Yaskawa INFORM job: SKRZYNIA_4040_0_STOPNI_2OBR.JBI

/JOB
//NAME SKRZYNIA_4040_0_STOPNI_2OBR
///FOLDERNAME 02-SKRZYNIE_JOBS
//POS
///NPOS 466,466,0,38,0,0
///TOOL 0
///POSTYPE PULSE
///PULSE
C00000=1055,-24125,84372,288,19725,204
C00001=0,-15438,65714,0,-68532,0
C00002=4718,-16587,59952,3396,-65485,-935
C00003=32997,-21499,42555,27623,-61436,21376
C00004=31759,-20688,42932,26837,-60850,21559
C00005=28987,-21156,42712,24818,-60442,22222
C00006=33447,-21964,42352,27886,-61721,21330
C00007=37687,-23357,41794,30651,-63289,20620
C00008=38979,-19018,48057,32961,-64962,20678
C00009=37261,-18075,48526,31902,-64209,20901
C00010=35830,-17198,48994,31015,-63571,21092
C00011=34080,-17614,48768,29780,-63290,21485
C00012=37261,-18075,48526,31902,-64209,20901
C00013=47373,-21912,40596,41149,-66086,26950
C00014=45033,-20851,41104,39798,-65001,27223
C00015=42790,-19693,41704,38494,-63946,27495
C00016=41070,-20182,41442,37324,-63566,27891
C00017=45033,-20851,41104,39798,-65001,27223
C00018=59624,-29540,14278,64846,-60867,16042
C00019=59624,-29540,14278,64846,-60867,16042
C00020=57357,-28542,14780,63940,-59509,16120
C00021=56188,-29140,14476,63237,-58995,16387
C00022=59588,-29370,14363,64862,-60819,16012
C00023=70875,-38414,-12574,117781,-105744,5605
C00024=70875,-38414,-12574,117781,-105744,5605
C00025=58486,-39981,-10562,86359,-50427,5279
C00026=56769,-35832,-2792,84059,-49443,6631
C00027=55152,-35009,-2405,83835,-48426,6454
C00028=53661,-35722,-2740,83085,-47530,6682
C00029=56769,-35832,-2792,84059,-49443,6631
C00030=45044,-23015,37260,35797,-71879,25522
C00031=39973,-29571,18873,35060,-63052,24165
C00032=38620,-28701,19269,34339,-62304,24363
C00033=36409,-29254,19014,32896,-61805,24958
C00034=44451,-29039,21934,37281,-65892,23702
C00035=49472,-39353,6917,53118,-50908,20251
C00036=45058,-39356,3832,51653,-47640,20099
C00037=42883,-38319,4163,50577,-46309,20295
C00038=40255,-38926,3967,48502,-45334,21060
C00039=46774,-39679,3737,52663,-48537,19827
C00040=48708,-40455,3517,53615,-49689,19657
C00041=43798,-39237,3871,50850,-47027,20335
C00042=41951,-38324,4161,49930,-45891,20507
C00043=39836,-38844,3994,48234,-45126,21137
C00044=48489,-40338,3551,53521,-49551,19665
C00045=41144,-42823,8332,45214,-41270,16613
C00046=27655,-47386,17113,29958,-26061,11007
C00047=27657,-47383,17112,100898,-60101,11012
C00048=27657,-47383,17112,100898,-60101,11012
C00049=48489,-40338,3551,53521,-49551,19665
C00050=44432,-39026,3936,51363,-47247,20139
C00051=42487,-38069,4248,50403,-46050,20315
C00052=39061,-38795,4009,47695,-44769,21310
C00053=44432,-39026,3936,51363,-47247,20139
C00054=43521,-36748,12770,50182,-45701,23408
C00055=41846,-35383,13175,49516,-44517,23399
C00056=39971,-34448,13485,48491,-43408,23582
C00057=37453,-34980,13306,46330,-42542,24334
C00058=41846,-35383,13175,49516,-44517,23399
C00059=78369,-41260,16071,67181,-65880,21417
C00060=137,-45861,52341,97,-67596,-14
C00061=11549,-53044,26255,3918,7271,6746
C00062=11549,-23006,80296,3918,7271,6746
C00063=11549,-23006,80296,3918,7271,6746
C00064=57941,-59676,-5815,65032,-36778,-7179
C00065=75493,-63502,-64712,103874,-64610,-6298
C00066=48206,-58699,-62794,109567,-46310,-10557
C00067=43841,-59955,-65018,113836,-43076,-9157
C00068=55379,-67378,-68041,108237,-48773,-4935
C00069=60826,-65014,-65501,105394,-54241,-6755
C00070=28458,-37240,33167,37371,-31902,2053
C00071=0,-44704,54767,0,2714,0
C00072=1055,-24125,84372,288,19725,204
C00073=0,-15438,65714,0,-68532,0
C00074=0,-15438,65714,966,-70097,42926
C00075=69988,-9219,57065,61610,-82752,27767
C00076=63113,-6157,59685,58080,-79692,28271
C00077=46291,-7558,63674,40492,-74068,29264
C00078=49370,-5991,66013,43448,-75651,29403
C00079=53417,-8187,64183,45775,-77170,28968
C00080=63113,-6157,59685,58080,-79692,28271
C00081=69988,-9219,57065,61610,-82752,27767
C00082=0,-15438,65714,966,-70097,42926
C00083=0,-15438,65714,0,-68532,0
C00084=1055,-24125,84372,288,19725,204
C00085=1055,-24125,84372,288,19725,204
C00086=0,-39065,65718,0,-582,0
C00087=0,-52280,40443,0,6876,0
C00088=0,-52280,40443,0,-40718,0
C00089=32359,-35955,27464,28918,-49457,29587
C00090=33244,-30989,28192,31082,-46894,28340
C00091=17628,-48691,-23897,104192,-11544,-8124
C00092=21099,-27494,32719,20191,-44662,31889
C00093=19639,-57374,-33308,34145,-23745,23766
C00094=18827,-52926,-25525,21842,-34932,29033
C00095=29904,-46498,-2819,27004,-47536,28031
C00096=45803,-31685,22885,64496,-39050,18987
C00097=0,-52277,40442,0,6872,2
///LIMIT ON
C00098=0,-38538,66749,0,-898,0
///LIMIT OFF
C00099=0,-52280,40443,0,-79033,35417
C00100=63837,-43435,-10267,65210,-58810,8342
C00101=51738,-38814,-970,57660,-53573,11589
C00102=47428,-40359,-5192,59734,-48299,10261
C00103=46171,-27309,20504,44749,-62331,18276
C00104=53914,-29436,22058,48262,-67266,17843
C00105=0,-52280,40443,0,-79033,35417
C00106=0,-38922,70509,0,-71891,28081
C00107=0,-38922,70509,0,-71891,28081
C00108=36958,-10079,72709,30464,-66560,20948
C00109=30104,-8063,72255,25983,-63748,21599
C00110=5528,-37153,828,214,-53033,28566
C00111=13946,-45192,10090,9828,-39459,25958
///LIMIT ON
C00112=404,-42897,57020,-1574,2523,869
///LIMIT OFF
C00113=0,-52280,40443,0,6876,0
C00114=-99253,-13690,44082,59847,13407,-31313
C00115=-87814,-12734,20141,45739,-14352,-64418
C00116=-86669,-6582,30812,41148,-16781,-62025
C00117=-85055,-5827,31548,44003,-17420,-63187
C00118=-85971,-6262,31124,42409,-17052,-62539
C00119=-86650,-5303,32069,41395,-16716,-62141
C00120=-94954,-14494,-1860,-7818,15857,-59130
C00121=-94509,1544,30797,-849,15127,-60471
C00122=-94509,4151,37772,-1041,12286,-60378
C00123=-88011,-10036,27574,37950,-16527,-60658
C00124=-86125,-12470,22545,29004,-25567,-58412
C00125=-85732,-21202,11427,30682,-24763,-59235
C00126=-84150,-10929,23786,31981,-25941,-59678
C00127=-83036,-10419,24246,33504,-26268,-60308
C00128=-84150,-10929,23786,31981,-25941,-59678
C00129=-85291,-9507,25078,30650,-25411,-59154
C00130=-84150,-10929,23786,31981,-25941,-59678
C00131=-85786,-16909,14677,31743,-23900,-59790
C00132=-84150,-10498,24888,31517,-26306,-59436
C00133=-83174,-10052,25293,32841,-26587,-59984
C00134=-84150,-10498,24888,31517,-26306,-59436
C00135=-85258,-9112,26156,30226,-25800,-58928
C00136=-84150,-10498,24888,31517,-26306,-59436
C00137=-87841,-18519,13420,28367,-23534,-58339
C00138=-84150,-10465,24972,31484,-26336,-59417
C00139=-83241,-10052,25348,32714,-26598,-59924
C00140=-84150,-10465,24972,31484,-26336,-59417
C00141=-85145,-9228,26102,30329,-25881,-58963
C00142=-84150,-10465,24972,31484,-26336,-59417
C00143=-86371,-18277,13606,30568,-23951,-59265
C00144=-84345,-11688,21985,32461,-25312,-59957
C00145=-83211,-11173,22442,34044,-25650,-60618
C00146=-84345,-11688,21985,32461,-25312,-59957
C00147=-85283,-10526,23025,31366,-24861,-59525
C00148=-84345,-11688,21985,32461,-25312,-59957
C00149=-86191,-19647,12567,30467,-24278,-59187
C00150=-84345,-10877,24073,31552,-26006,-59481
C00151=-83051,-10286,24607,33321,-26381,-60213
C00152=-84345,-10877,24073,31552,-26006,-59481
C00153=-85179,-9842,25009,30582,-25619,-59100
C00154=-84345,-10877,24073,31552,-26006,-59481
C00155=-85438,-18022,14839,31140,-24818,-59429
C00156=-84247,-11820,22550,32049,-25753,-59727
C00157=-84104,-10976,23642,32111,-25899,-59738
C00158=-82990,-10465,24105,33639,-26227,-60372
C00159=-84104,-10976,23642,32111,-25899,-59738
C00160=-84898,-9998,24525,31196,-25529,-59378
C00161=-84104,-10976,23642,32111,-25899,-59738
C00162=-86610,-16845,14732,30573,-23614,-59301
C00163=-84104,-10864,23927,31990,-25993,-59674
C00164=-82824,-10273,24459,33737,-26370,-60397
C00165=-84104,-10864,23927,31990,-25993,-59674
C00166=-84789,-10021,24690,31200,-25673,-59363
C00167=-84104,-10864,23927,31990,-25993,-59674
C00168=-83806,-19585,12613,33764,-25080,-60559
C00169=-83924,-10205,25475,31619,-26533,-59453
C00170=-82780,-9675,25960,33156,-26866,-60087
C00171=-83924,-10205,25475,31619,-26533,-59453
C00172=-84478,-9530,26093,30986,-26280,-59206
C00173=-83924,-10205,25475,31619,-26533,-59453
C00174=-87149,-17993,13826,29513,-23647,-58830
C00175=-84920,-13182,20975,31162,-25481,-59361
C00176=-83711,-10572,24852,32056,-26475,-59649
C00177=-82779,-10142,25241,33309,-26748,-60166
C00178=-83711,-10572,24852,32056,-26475,-59649
C00179=-84370,-9774,25579,31305,-26170,-59356
C00180=-83711,-10572,24852,32056,-26475,-59649
C00181=-83642,-3679,42021,23358,-36761,-56118
C00182=-85886,-5975,41264,18964,-40261,-54782
C00183=-83919,-11632,22322,32811,-25616,-60079
C00184=-82884,-11162,22742,34234,-25925,-60671
C00185=-83919,-11632,22322,32811,-25616,-60079
C00186=-84723,-10654,23196,31887,-25230,-59715
C00187=-83919,-11632,22322,32811,-25616,-60079
C00188=-87348,-16035,7353,17528,-35245,-56477
C00189=-86244,-15062,8172,18754,-35315,-57058
C00190=-86244,-16649,3638,19674,-33501,-57585
C00191=-85308,-16228,3988,20718,-33648,-58082
C00192=-86244,-16649,3638,19674,-33501,-57585
C00193=-86740,-15973,4201,19194,-33277,-57362
C00194=-86244,-16649,3638,19674,-33501,-57585
C00195=-73780,-8639,20128,34258,-51705,-52097
C00196=-90711,-17528,-28778,11328,-28245,-57111
C00197=-92565,-19610,-33223,7138,-24591,-57051
C00198=-91512,-19116,-32812,8551,-24603,-57834
C00199=-92565,-19610,-33223,7138,-24591,-57051
C00200=-93003,-18716,-32476,6600,-24397,-56752
C00201=-92565,-19610,-33223,7138,-24591,-57051
C00202=-92565,-19610,-33223,7138,-24591,-57051
C00203=-95836,-54375,-51122,6031,-17685,-48210
C00204=-95836,-54375,-51122,6031,-17685,-48210
C00205=-71303,-59965,-23787,8701,20788,-26710
C00206=-43821,-47238,-2775,-3022,56549,-3681
C00207=-20126,-26882,59542,2406,16879,-9162
C00208=-20126,-26882,59542,2406,16879,-9162
C00209=98601,-10520,92678,4674,-40855,-9615
C00210=95537,-19831,-2695,-2933,-44471,35837
C00211=92548,-20391,-28429,-6186,-30623,55200
C00212=91429,-17018,-28974,-8057,-27827,56250
C00213=91429,-17018,-28974,-8057,-27827,56250
C00214=90371,-16495,-28521,-9286,-27856,56953
C00215=91429,-17018,-28974,-8057,-27827,56250
C00216=92033,-15799,-27911,-7415,-27588,55880
C00217=91429,-17018,-28974,-8057,-27827,56250
C00218=92548,-20391,-28429,-6186,-30623,55200
C00219=91156,-15018,-4648,-8036,-38181,54813
C00220=90585,-14766,-4428,-8565,-38201,55100
C00221=88830,-13959,-3717,-10186,-38284,55977
C00222=89897,-14456,-4157,-9202,-38230,55445
C00223=90761,-12944,-2809,-8452,-37927,55043
C00224=89897,-14456,-4157,-9202,-38230,55445
C00225=89670,-8466,73559,-9449,-60959,55261
C00226=89910,-11217,67535,-9455,-58896,55399
C00227=85786,-16735,14816,-31782,-23869,59812
C00228=83514,-12996,17929,-35760,-24132,61552
C00229=82251,-12406,18443,-37550,-24551,62308
C00230=83514,-12996,17929,-35760,-24132,61552
C00231=84258,-12095,18717,-34917,-23742,61217
C00232=83514,-12996,17929,-35760,-24132,61552
C00233=87149,-17993,13826,-29513,-23647,58830
C00234=83118,-12818,18089,-36330,-24263,61791
C00235=81915,-12248,18589,-38020,-24666,62504
C00236=83118,-12818,18089,-36330,-24263,61791
C00237=83897,-11882,18912,-35460,-23856,61445
C00238=83118,-12818,18089,-36330,-24263,61791
C00239=83806,-19585,12613,-33764,-25080,60559
C00240=82998,-13006,17925,-36445,-24332,61826
C00241=81675,-12378,18472,-38297,-24777,62607
C00242=82998,-13006,17925,-36445,-24332,61826
C00243=83876,-11958,18841,-35466,-23874,61442
C00244=82998,-13006,17925,-36445,-24332,61826
C00245=86610,-16845,14732,-30573,-23614,59301
C00246=82493,-13239,17725,-37070,-24559,62089
C00247=81406,-12724,18174,-38578,-24928,62723
C00248=82493,-13239,17725,-37070,-24559,62089
C00249=83436,-12134,18690,-36041,-24064,61684
C00250=82493,-13239,17725,-37070,-24559,62089
C00251=84814,-16043,15376,-33312,-24093,60464
C00252=82555,-13613,17404,-36910,-24580,62015
C00253=81384,-13062,17878,-38534,-24974,62698
C00254=82555,-13613,17404,-36910,-24580,62015
C00255=83566,-12434,18427,-35805,-24047,61580
C00256=82555,-13613,17404,-36910,-24580,62015
C00257=86191,-19647,12567,-30467,-24278,59187
C00258=82500,-13648,17375,-36975,-24607,62039
C00259=81467,-13161,17792,-38413,-24955,62645
C00260=82500,-13648,17375,-36975,-24607,62039
C00261=83481,-12505,18364,-35905,-24087,61617
C00262=82500,-13648,17375,-36975,-24607,62039
C00263=86371,-18277,13606,-30568,-23951,59265
C00264=82904,-13790,17251,-36416,-24470,61808
C00265=81715,-13237,17726,-38081,-24865,62509
C00266=82904,-13790,17251,-36416,-24470,61808
C00267=83686,-12878,18037,-35556,-24055,61469
C00268=82904,-13790,17251,-36416,-24470,61808
C00269=87841,-18519,13420,-28367,-23534,58339
C00270=82748,-13879,17174,-36603,-24542,61883
C00271=81692,-13388,17594,-38077,-24893,62505
C00272=82748,-13879,17174,-36603,-24542,61883
C00273=83607,-12881,18032,-35663,-24082,61515
C00274=82748,-13879,17174,-36603,-24542,61883
C00275=85786,-16909,14677,-31743,-23900,59790
C00276=82520,-14198,16902,-36833,-24674,61972
C00277=81460,-13708,17319,-38301,-25026,62591
C00278=82520,-14198,16902,-36833,-24674,61972
C00279=83571,-12989,17938,-35691,-24113,61524
C00280=82520,-14198,16902,-36833,-24674,61972
C00281=85732,-21202,11427,-30682,-24763,59235
C00282=82398,-14365,16763,-36952,-24745,62014
C00283=81172,-13798,17245,-38643,-25153,62725
C00284=82398,-14365,16763,-36952,-24745,62014
C00285=83600,-12984,17944,-35650,-24102,61504
C00286=82398,-14365,16763,-36952,-24745,62014
C00287=86140,-12802,12665,-93523,-10743,85795
C00288=86140,-12802,12665,-93523,-10743,85795
C00289=85030,-12289,13120,-93723,-11463,85776
C00290=86140,-12802,12665,-93523,-10743,85795
C00291=86958,-11660,13681,-94506,-10238,86349
C00292=85239,-16743,-4327,42764,21357,45785
C00293=86674,107,23869,25042,24033,51593
C00294=86674,2327,30134,27824,21680,50173
C00295=87715,-15254,10554,-91589,-9692,85040
C00296=85045,-36869,-4353,-28502,-22832,52282
C00297=0,-24029,84339,0,19981,0
C00298=0,-24029,84339,0,19981,0
C00299=3172,-24246,80980,3465,15913,689
C00300=-86563,-26985,13879,10257,-21548,-45530
C00301=-86191,-19647,12567,30467,-24278,-59187
C00302=-83221,-13587,17636,37793,-25116,-62228
C00303=-91978,-13833,14560,12391,-18633,-51524
C00304=-94992,-13830,14285,1276,-18012,-46664
C00305=-84074,-17488,11256,38660,-23649,-62784
C00306=-73679,-33270,1000,44272,-31600,-64253
///LIMIT ON
C00307=-86926,-60758,23267,6576,1160,-9545
///LIMIT OFF
C00308=0,-52280,40443,0,6876,0
///LIMIT ON
C00309=82475,-58079,26734,835,4084,4444
///LIMIT OFF
C00310=97932,-26840,7691,8784,-23444,42538
C00311=87166,-16607,16322,-25365,-24201,56345
C00312=84699,-11354,21752,-29145,-24735,57949
C00313=84804,-11023,22730,-28561,-25071,57659
C00314=85100,-26994,10417,-24982,-28140,55821
C00315=0,-52280,40443,0,6876,0
C00316=0,-52280,40443,0,6876,0
///LIMIT ON
C00317=-90140,-60305,18108,-2708,1721,-7625
///LIMIT OFF
C00318=-95594,-27428,6866,-4663,-19832,-42154
C00319=-98688,-13767,16447,-18366,-10080,-35766
C00320=-98967,-3050,34440,-28957,-8622,-29685
C00321=-100063,5316,51567,-32262,-10006,-27560
C00322=-94586,18541,64268,-6451,10518,-43578
C00323=-95535,2380,25473,239,27557,-47214
C00324=-91259,3120,34463,-5130,22041,-43946
C00325=-95333,12702,45733,36,21375,-47085
C00326=-99268,-13088,27343,-18620,-14105,-35021
///LIMIT ON
C00327=-90140,-60305,18108,-2708,1721,-7625
///LIMIT OFF
C00328=0,-52280,40443,0,6876,0
///LIMIT ON
C00329=84259,-57935,27522,-3761,3673,6310
///LIMIT OFF
C00330=86507,-39672,4297,-27618,-16640,46340
C00331=73669,-37119,-20783,-92053,-19719,85232
C00332=86539,-20830,1725,-71850,-11773,76853
C00333=90325,-18913,6238,-62161,-7452,70888
///LIMIT ON
C00334=97679,-11879,12650,-55334,4229,66281
///LIMIT OFF
C00335=98389,-8856,11720,-15676,14634,48538
C00336=96255,-748,20886,-3277,24061,38276
C00337=95132,-6008,10010,1655,28777,36730
C00338=94050,-4188,7205,-2481,41508,36662
C00339=98126,4908,16834,-5042,41918,38535
C00340=100487,-9453,-1206,-10413,41328,41147
C00341=96250,-19428,-8283,-4838,27297,37910
C00342=86507,-39672,4297,-27618,-16640,46340
///LIMIT ON
C00343=84259,-57935,27522,-3761,3673,6310
///LIMIT OFF
C00344=0,-52280,40443,0,6876,0
C00345=0,-27933,77061,0,20812,0
C00346=0,-27933,77061,0,20812,0
C00347=0,-52280,40443,0,6876,0
///LIMIT ON
C00348=-91970,-60791,14435,-3343,512,-9412
///LIMIT OFF
C00349=-98647,-24138,10005,-11519,-21203,-39749
C00350=-99883,-13980,22886,-11640,-25090,-40341
C00351=-99702,-9154,61728,-1148,-61809,-40243
C00352=-84328,-13042,29707,23458,-33731,-54641
C00353=-83230,-4243,39143,25752,-34754,-55611
C00354=-83186,-4481,38540,26056,-34403,-55733
C00355=-76259,-18287,26646,31659,-38322,-57579
C00356=-89741,-28009,12101,4461,-28076,-46404
///LIMIT ON
C00357=-91970,-60791,14435,-3343,512,-9412
///LIMIT OFF
C00358=0,-52280,40443,0,6876,0
///LIMIT ON
C00359=91083,-60784,14823,-9043,-825,15173
///LIMIT OFF
C00360=83869,-19403,12921,-33769,-24740,60260
C00361=83869,-19403,12921,-33769,-24740,60260
C00362=83932,-19538,53415,-33663,-71112,60249
C00363=83932,-19538,53415,-33663,-71112,60249
C00364=82480,-12247,21118,-35440,-26416,60009
C00365=82411,-11538,19708,-37356,-25248,61001
C00366=82612,-9723,24389,-34866,-26650,59727
C00367=79790,-20261,14917,-36681,-28829,60258
C00368=76554,-29711,-1870,-46042,-25952,65654
///LIMIT ON
C00369=91083,-60784,14823,-9043,-825,15173
///LIMIT OFF
C00370=0,-52280,40443,0,6876,0
///LIMIT ON
C00371=-91526,-60598,16699,7584,176,-13289
///LIMIT OFF
C00372=-81382,-25890,9219,35455,-25500,-59095
C00373=-86453,-20958,12525,30076,-22568,-57089
C00374=-86589,-16097,16237,31250,-21582,-57704
C00375=-98933,-11298,20505,-13970,-18736,-37953
C00376=-98281,-10965,21163,-11559,-18548,-39330
C00377=-85424,-18472,14402,34409,-22969,-58895
C00378=-74746,-27148,8488,44263,-29128,-62418
C00379=-81326,-27507,8265,35533,-26282,-59001
///LIMIT ON
C00380=-91415,-60262,16631,7870,-73,-13734
///LIMIT OFF
C00381=24,-24029,84339,7,19981,5
C00382=100404,-52373,45687,-1822,14816,-5144
C00383=75939,-26469,7919,-40869,-29645,63133
C00384=81882,-22565,10470,-35355,-26404,61107
C00385=82801,-12246,21732,-34208,-26055,60642
C00386=91824,-10567,23615,-8659,-22197,49820
C00387=96485,-9539,26282,5686,-23135,43736
C00388=77262,-23244,14300,-38922,-31295,61912
C00389=96357,-33562,33410,58602,-23427,10353
C00390=568,-24029,84339,168,19981,112
///LIMIT ON
C00391=-91970,-60791,14435,-3343,512,-9412
///LIMIT OFF
C00392=-98991,-22833,11519,-12824,-17638,-36336
C00393=-86376,-13627,18436,38326,-18406,-58533
C00394=-85581,-10814,20279,41280,-18093,-59893
C00395=-85559,-10490,20860,41006,-18219,-59754
C00396=-86274,-24518,9978,34497,-20333,-56613
C00397=-91684,-53777,2301,20525,-9313,-33684
C00398=-67305,-55044,34987,1504,5690,-2468
C00399=0,-52280,40443,0,6876,0
///LIMIT ON
C00400=77036,-56616,31288,-2531,4707,4197
///LIMIT OFF
C00401=84359,-28321,8817,-32860,-20485,54199
C00402=81156,-16932,14874,-39538,-26422,62851
C00403=93321,-15690,11640,-5466,-17578,48664
C00404=91343,-14550,14673,-11914,-19185,51366
C00405=77970,-27630,4721,-41834,-28549,63607
C00406=81111,-35571,7141,-33980,-21909,52006
///LIMIT ON
C00407=82490,-55811,26416,-6832,1088,10458
///LIMIT OFF
C00408=0,-52280,40443,0,6876,0
C00409=0,-28135,76691,0,20839,0
C00410=0,-28135,76691,0,20839,0
C00411=-45332,-39712,59352,-1730,18713,2903
C00412=-94065,-8316,59352,-1730,-37754,-40387
C00413=-100331,-14895,33931,-8215,-36518,-40227
C00414=-98931,-8578,39429,-6260,-48307,-43744
C00415=-100336,-4176,46216,-7600,-55875,-44633
C00416=-93952,8947,73671,995,-68520,-43850
C00417=-98791,-3170,32594,-4861,-60761,-43748
C00418=-98723,4324,37855,-4919,-58743,-43677
C00419=-98691,-12730,-17828,-7584,-33364,-41886
C00420=-98599,-14408,-28132,-8909,-27584,-41168
C00421=-99605,-15546,-21493,-8548,-33053,-41326
C00422=-98632,914,40428,-4141,-58435,-42510
C00423=-93952,8947,73671,995,-68520,-43850
C00424=-88754,54,62805,4404,-67858,-45120
C00425=-100222,-4532,45667,-7492,-55263,-44561
C00426=-100331,-14895,33931,-8215,-36518,-40227
C00427=-94065,-8316,59352,-1730,-37754,-40387
C00428=-45544,-32973,71870,-2133,15168,3033
C00429=0,-28135,76691,0,20839,0
C00430=54178,-17846,77779,596,-29686,20997
C00431=54178,-17846,77779,596,-29686,20997
C00432=99462,-18987,75418,611,-28919,20989
C00433=98707,-9390,78674,1080,-71212,38250
C00434=98768,-5182,41096,1808,-44974,38308
C00435=100431,1771,51615,3823,-56746,39115
C00436=97953,-6621,17555,2289,-50176,39420
C00437=95834,-5353,18817,760,-50052,40242
C00438=86579,-3733,19265,-13263,-48799,44764
C00439=89140,-11519,-8899,-11291,-36869,46482
C00440=89026,-14065,-21014,-13447,-30614,47708
C00441=90457,-16080,-12990,-9972,-37305,45724
C00442=97953,-6621,17555,2289,-50176,39420
C00443=100431,1771,51615,3823,-56746,39115
C00444=98768,-5182,41096,1808,-44974,38308
C00445=98707,-9390,78674,1080,-71212,38250
C00446=0,-28135,76691,0,20839,0
C00447=0,-28135,76691,0,20839,0
///LIMIT ON
C00448=-91526,-60598,16699,7584,176,-13289
///LIMIT OFF
C00449=-81382,-25890,9219,35455,-25500,-59095
C00450=-81382,-25890,9219,35455,-25500,-59095
C00451=-85509,-13950,19358,32213,-22393,-58041
C00452=-96341,-12327,18855,-5124,-17594,-42111
C00453=-97523,-9822,24708,-8570,-19966,-40659
C00454=-84656,-25369,12054,31249,-26195,-57129
///LIMIT ON
C00455=-82652,-57346,29982,2770,3944,-5064
///LIMIT OFF
C00456=0,-52280,40443,0,6876,0
C00457=60653,-54633,35892,-1212,5841,2035
C00458=77942,-28227,6869,-38010,-29303,61907
C00459=82500,-13648,17375,-36975,-24607,62039
C00460=80731,-11587,18684,-41654,-25449,63953
C00461=80409,-10373,22284,-40214,-26848,63104
C00462=64389,-31987,5108,-50419,-37074,66126
C00463=60653,-54633,35892,-1212,5841,2035
C00464=0,-52280,40443,0,6876,0
C00465=0,-28167,76633,0,20843,0
BC00000=320972
BC00001=320972
BC00002=295997
BC00003=264574
BC00004=264574
BC00005=264574
BC00006=264574
BC00007=264574
BC00008=315010
BC00009=315010
BC00010=315010
BC00011=315010
BC00012=315010
BC00013=387267
BC00014=387267
BC00015=387267
BC00016=387267
BC00017=387267
BC00018=438071
BC00019=438071
BC00020=438071
BC00021=438071
BC00022=438071
BC00023=392105
BC00024=508747
BC00025=486795
BC00026=486795
BC00027=486795
BC00028=486795
BC00029=486795
BC00030=597036
BC00031=597036
BC00032=597036
BC00033=597036
BC00034=597036
BC00035=634297
BC00036=634297
BC00037=634297
BC00038=634297
BC00039=634297
BC00040=684103
BC00041=680754
BC00042=680754
BC00043=680754
BC00044=680754
BC00045=597007
BC00046=614958
BC00047=614956
BC00048=689447
BC00049=767343
BC00050=758255
BC00051=758255
BC00052=758255
BC00053=758255
BC00054=788049
BC00055=778832
BC00056=778832
BC00057=778832
BC00058=778832
BC00059=788230
BC00060=758518
BC00061=641445
BC00062=641445
BC00063=507948
BC00064=642386
BC00065=658668
BC00066=658671
BC00067=717186
BC00068=719761
BC00069=632565
BC00070=557994
BC00071=591569
BC00072=320972
BC00073=320972
BC00074=320972
BC00075=316460
BC00076=316460
BC00077=316587
BC00078=256438
BC00079=255226
BC00080=316460
BC00081=316460
BC00082=320972
BC00083=320972
BC00084=320972
BC00085=413336
BC00086=595855
BC00087=671091
BC00088=717147
BC00089=791187
BC00090=791187
BC00091=791187
BC00092=787699
BC00093=791187
BC00094=791187
BC00095=791187
BC00096=752948
BC00097=678155
BC00098=415650
BC00099=415650
BC00100=453835
BC00101=453835
BC00102=453835
BC00103=400874
BC00104=399813
BC00105=415650
BC00106=415650
BC00107=553692
BC00108=553692
BC00109=553595
BC00110=553692
BC00111=553692
BC00112=494617
BC00113=645849
BC00114=677569
BC00115=779301
BC00116=779301
BC00117=779301
BC00118=779301
BC00119=779301
BC00120=779301
BC00121=779301
BC00122=779301
BC00123=779301
BC00124=779301
BC00125=810022
BC00126=803206
BC00127=803206
BC00128=803206
BC00129=803206
BC00130=803206
BC00131=748578
BC00132=748578
BC00133=748578
BC00134=748578
BC00135=748578
BC00136=748578
BC00137=687134
BC00138=679166
BC00139=679166
BC00140=679166
BC00141=679166
BC00142=679166
BC00143=625689
BC00144=625689
BC00145=625689
BC00146=625689
BC00147=625689
BC00148=625689
BC00149=564239
BC00150=557007
BC00151=557007
BC00152=557007
BC00153=557007
BC00154=557007
BC00155=502795
BC00156=502795
BC00157=502795
BC00158=502795
BC00159=502795
BC00160=502795
BC00161=502795
BC00162=441351
BC00163=433063
BC00164=433063
BC00165=433063
BC00166=433063
BC00167=433063
BC00168=379907
BC00169=379907
BC00170=379907
BC00171=379907
BC00172=379907
BC00173=379907
BC00174=318463
BC00175=313496
BC00176=310802
BC00177=310802
BC00178=310802
BC00179=310802
BC00180=310802
BC00181=310802
BC00182=257020
BC00183=257020
BC00184=257020
BC00185=257020
BC00186=257020
BC00187=257020
BC00188=367191
BC00189=367191
BC00190=367191
BC00191=367191
BC00192=367191
BC00193=367191
BC00194=367191
BC00195=398324
BC00196=367601
BC00197=367601
BC00198=367601
BC00199=367601
BC00200=367601
BC00201=367601
BC00202=456025
BC00203=456025
BC00204=545675
BC00205=514634
BC00206=493841
BC00207=450584
BC00208=482012
BC00209=515684
BC00210=426185
BC00211=369502
BC00212=369502
BC00213=369502
BC00214=369502
BC00215=369502
BC00216=369502
BC00217=369502
BC00218=400224
BC00219=399607
BC00220=399607
BC00221=399607
BC00222=399607
BC00223=399607
BC00224=399607
BC00225=326898
BC00226=274752
BC00227=257020
BC00228=261075
BC00229=261075
BC00230=261075
BC00231=261075
BC00232=261075
BC00233=318463
BC00234=316969
BC00235=316969
BC00236=316969
BC00237=316969
BC00238=316969
BC00239=379907
BC00240=383960
BC00241=383960
BC00242=383960
BC00243=383960
BC00244=383960
BC00245=441351
BC00246=440478
BC00247=440478
BC00248=440478
BC00249=440478
BC00250=440478
BC00251=502795
BC00252=507822
BC00253=507822
BC00254=507822
BC00255=507822
BC00256=507822
BC00257=564239
BC00258=561088
BC00259=561088
BC00260=561088
BC00261=561088
BC00262=561088
BC00263=625689
BC00264=629404
BC00265=629404
BC00266=629404
BC00267=629404
BC00268=629404
BC00269=687134
BC00270=685797
BC00271=685797
BC00272=685797
BC00273=685797
BC00274=685797
BC00275=748578
BC00276=751644
BC00277=751644
BC00278=751644
BC00279=751644
BC00280=751644
BC00281=810022
BC00282=807962
BC00283=807962
BC00284=807962
BC00285=807962
BC00286=807962
BC00287=781157
BC00288=781157
BC00289=781157
BC00290=781157
BC00291=781157
BC00292=781157
BC00293=781157
BC00294=781157
BC00295=781157
BC00296=747172
BC00297=631717
BC00298=631717
BC00299=536262
BC00300=587497
BC00301=629276
BC00302=629276
BC00303=629273
BC00304=689316
BC00305=689722
BC00306=689722
BC00307=689722
BC00308=689722
BC00309=676777
BC00310=626309
BC00311=626309
BC00312=626309
BC00313=686147
BC00314=666866
BC00315=535311
BC00316=654423
BC00317=654423
BC00318=763863
BC00319=763863
BC00320=756369
BC00321=783031
BC00322=765866
BC00323=772343
BC00324=772343
BC00325=772343
BC00326=765867
BC00327=608340
BC00328=654423
BC00329=654423
BC00330=749197
BC00331=771932
BC00332=771932
BC00333=777363
BC00334=772686
BC00335=795648
BC00336=789230
BC00337=788718
BC00338=787466
BC00339=787628
BC00340=771932
BC00341=771932
BC00342=703114
BC00343=700506
BC00344=700506
BC00345=608083
BC00346=454048
BC00347=454048
BC00348=454045
BC00349=454045
BC00350=314610
BC00351=314610
BC00352=260095
BC00353=233578
BC00354=314100
BC00355=314100
BC00356=399390
BC00357=454045
BC00358=454048
BC00359=454048
BC00360=415438
BC00361=318616
BC00362=337524
BC00363=283281
BC00364=258308
BC00365=239237
BC00366=316196
BC00367=316492
BC00368=415438
BC00369=454048
BC00370=454048
BC00371=424591
BC00372=499643
BC00373=499643
BC00374=499643
BC00375=499017
BC00376=558187
BC00377=558372
BC00378=558372
BC00379=491837
BC00380=423635
BC00381=427852
BC00382=427852
BC00383=498431
BC00384=500914
BC00385=500914
BC00386=500914
BC00387=560290
BC00388=560393
BC00389=502622
BC00390=341722
BC00391=454045
BC00392=738156
BC00393=738156
BC00394=738156
BC00395=784552
BC00396=798230
BC00397=706682
BC00398=706682
BC00399=706682
BC00400=706682
BC00401=740130
BC00402=752844
BC00403=752844
BC00404=800324
BC00405=790210
BC00406=726674
BC00407=656571
BC00408=648379
BC00409=434801
BC00410=242446
BC00411=242446
BC00412=242446
BC00413=258298
BC00414=258298
BC00415=267171
BC00416=267171
BC00417=267171
BC00418=267555
BC00419=267287
BC00420=267176
BC00421=267171
BC00422=267171
BC00423=267171
BC00424=267171
BC00425=266454
BC00426=258298
BC00427=242446
BC00428=242446
BC00429=242446
BC00430=242447
BC00431=377887
BC00432=409113
BC00433=242446
BC00434=242444
BC00435=257344
BC00436=273769
BC00437=273769
BC00438=273768
BC00439=256264
BC00440=256264
BC00441=256264
BC00442=273769
BC00443=257344
BC00444=242444
BC00445=242446
BC00446=242446
BC00447=420623
BC00448=424591
BC00449=434461
BC00450=374803
BC00451=374803
BC00452=374803
BC00453=432481
BC00454=433579
BC00455=433579
BC00456=433579
BC00457=433579
BC00458=381745
BC00459=381745
BC00460=381745
BC00461=440658
BC00462=441577
BC00463=433579
BC00464=433579
BC00465=433581
///POSTYPE BASE
///RECTAN
///RCONF 1,0,0,0,0,0,0,0,0,0,0,0,0,0,0,0,0,0,0,0,0,0,0,0
P00006=0.000,0.000,0.000,0.0000,0.0000,0.0000
///RCONF 0,0,0,0,0,0,0,0,0,0,0,0,0,0,0,0,0,0,0,0,0,0,0,0
P00057=0.000,0.000,2.000,0.0000,0.0000,0.0000
///RCONF 1,0,0,0,0,0,0,0,0,0,0,0,0,0,0,0,0,0,0,0,0,0,0,0
P00099=0.011,-2.380,1.226,0.0000,0.0000,0.0000
P00100=-0.081,2.558,4.482,0.0000,0.0000,0.0000
P00101=0.030,-2.286,2.993,0.0000,0.0000,0.0000
P00102=-0.005,-1.108,1.644,0.0000,0.0000,0.0000
P00103=-0.094,-3.400,4.200,0.0000,0.0000,0.0000
P00104=0.043,-2.127,5.826,0.0000,0.0000,0.0000
P00105=-0.043,0.662,5.286,0.0000,0.0000,0.0000
P00106=-0.018,-2.519,0.237,0.0000,0.0000,0.0000
P00107=-0.008,-4.537,-4.500,0.0000,0.0000,0.0000
P00108=0.014,-3.040,2.637,0.0000,0.0000,0.0000
///RCONF 0,0,0,0,0,0,0,0,0,0,0,0,0,0,0,0,0,0,0,0,0,0,0,0
P00299=-1.404,-0.874,9.133,0.0000,0.0000,0.0000
///RCONF 1,0,0,0,0,0,0,0,0,0,0,0,0,0,0,0,0,0,0,0,0,0,0,0
P00301=0.046,-2.112,7.779,0.0000,0.0000,0.0000
P00302=-0.180,-2.409,6.326,0.0000,0.0000,0.0000
///RCONF 0,0,0,0,0,0,0,0,0,0,0,0,0,0,0,0,0,0,0,0,0,0,0,0
P00303=-0.004,-1.437,-4.584,0.0000,0.0000,0.0000
P00304=0.028,-1.666,-4.234,0.0000,0.0000,0.0000
P00305=-0.003,-1.920,-3.501,0.0000,0.0000,0.0000
P00306=0.015,-2.252,-3.054,0.0000,0.0000,0.0000
P00307=0.019,-2.151,-5.077,0.0000,0.0000,0.0000
P00308=-0.003,-2.092,-4.888,0.0000,0.0000,0.0000
P00309=-0.040,-2.205,-4.992,0.0000,0.0000,0.0000
P00310=-0.006,-2.490,-5.925,0.0000,0.0000,0.0000
P00311=-0.007,-2.079,-5.307,0.0000,0.0000,0.0000
P00312=-0.032,2.202,-7.632,0.0000,0.0000,0.0000
///RCONF 1,0,0,0,0,0,0,0,0,0,0,0,0,0,0,0,0,0,0,0,0,0,0,0
P00349=0.060,0.167,-1.133,0.0000,0.0000,0.0000
///RCONF 0,0,0,0,0,0,0,0,0,0,0,0,0,0,0,0,0,0,0,0,0,0,0,0
P00350=11.519,-0.008,1.149,0.0000,0.0000,0.0000
P00351=13.563,-0.027,-0.653,0.0000,0.0000,0.0000
P00352=13.252,-0.027,-0.827,0.0000,0.0000,0.0000
P00353=10.971,-0.082,0.776,0.0000,0.0000,0.0000
P00354=-0.024,2.508,-1.824,0.0000,0.0000,0.0000
P00355=-0.001,2.528,-1.131,0.0000,0.0000,0.0000
P00356=-0.034,2.921,-0.262,0.0000,0.0000,0.0000
P00357=0.003,3.386,-0.091,0.0000,0.0000,0.0000
P00358=0.014,3.037,-0.020,0.0000,0.0000,0.0000
P00359=-0.005,2.731,0.912,0.0000,0.0000,0.0000
P00360=-0.011,3.412,0.438,0.0000,0.0000,0.0000
P00361=0.018,3.050,1.253,0.0000,0.0000,0.0000
//INST
///DATE 2025/03/28 09:07
///ATTR SC,RW
///GROUP1 RB1,BS1
NOP
CALL JOB:MOVE_INTO_TUNNEL
SFTOF
'------------------------
'------------------------
'SPOINA SRODEK DOL
'------------------------
'------------------------
MOVJ C00000 BC00000 VJ=10.00
MOVJ C00001 BC00001 VJ=30.00
SFTOF
MOVL C00002 BC00002 V=166.7
MOVL C00003 BC00003 V=166.7 PL=0
REFP 3 C00004 BC00004
CALL JOB:SEARCH-R1
IMOV P0057 V=23.0
SET P0099 P0006
SFTON P0099
REFP 3 C00005 BC00005
CALL JOB:SEARCH-R1
SET P0099 P0006
SFTON P0099
MOVL C00006 BC00006 V=166.7 PL=0
'TEST
SFTOF
MOVL C00007 BC00007 V=333.3
MOVL C00008 BC00008 V=333.3
'------------------------
'W38 L
'------------------------
'TEST
MOVL C00009 BC00009 V=166.7 PL=0
REFP 3 C00010 BC00010
CALL JOB:SEARCH-R1
IMOV P0057 V=23.0
SET P0100 P0006
SFTON P0100
REFP 3 C00011 BC00011
CALL JOB:SEARCH-R1
SET P0100 P0006
SFTON P0100
MOVL C00012 BC00012 V=166.7 PL=0
'TEST
SFTOF
MOVJ C00013 BC00013 VJ=20.00
'------------------------
'W45 P
'------------------------
MOVL C00014 BC00014 V=166.7 PL=0
REFP 3 C00015 BC00015
CALL JOB:SEARCH-R1
IMOV P0057 V=23.0
SET P0101 P0006
SFTON P0101
REFP 3 C00016 BC00016
CALL JOB:SEARCH-R1
SET P0101 P0006
SFTON P0101
MOVL C00017 BC00017 V=166.7 PL=0
'TEST
SFTOF
MOVJ C00018 BC00018 VJ=20.00
'------------------------
'W45 L
'------------------------
MOVL C00019 BC00019 V=133.3 PL=0
REFP 3 C00020 BC00020
CALL JOB:SEARCH-R1
IMOV P0057 V=23.0
SET P0102 P0006
SFTON P0102
REFP 3 C00021 BC00021
CALL JOB:SEARCH-R1
SET P0102 P0006
SFTON P0102
MOVL C00022 BC00022 V=250.0 PL=0
'TEST
SFTOF
MOVJ C00023 BC00023 VJ=30.00
MOVJ C00024 BC00024 VJ=30.00
MOVJ C00025 BC00025 VJ=20.00
'------------------------
'W48 P
'------------------------
'TEST
MOVL C00026 BC00026 V=133.3 PL=0
REFP 3 C00027 BC00027
CALL JOB:SEARCH-R1
IMOV P0057 V=23.0
SET P0103 P0006
SFTON P0103
REFP 3 C00028 BC00028
CALL JOB:SEARCH-R1
SET P0103 P0006
SFTON P0103
MOVL C00029 BC00029 V=166.7 PL=0
'TEST
SFTOF
MOVL C00030 BC00030 V=250.0
'------------------------
'W48 L
'------------------------
SFTOF
MOVL C00031 BC00031 V=133.3 PL=0
REFP 3 C00032 BC00032
CALL JOB:SEARCH-R1
IMOV P0057 V=23.0
SET P0104 P0006
SFTON P0104
REFP 3 C00033 BC00033
CALL JOB:SEARCH-R1
SET P0104 P0006
SFTON P0104
MOVL C00034 BC00034 V=166.7 PL=0
SFTOF
MOVJ C00035 BC00035 VJ=20.00
'------------------------
'W36 P
'------------------------
MOVL C00036 BC00036 V=133.3 PL=0
REFP 3 C00037 BC00037
CALL JOB:SEARCH-R1
IMOV P0057 V=23.0
SET P0105 P0006
SFTON P0105
REFP 3 C00038 BC00038
CALL JOB:SEARCH-R1
SET P0105 P0006
SFTON P0105
MOVL C00039 BC00039 V=166.7 PL=0
'TEST
SFTOF
MOVJ C00040 BC00040 VJ=20.00
'------------------------
'W36 L
'------------------------
MOVL C00041 BC00041 V=166.7 PL=0
REFP 3 C00042 BC00042
CALL JOB:SEARCH-R1
IMOV P0057 V=23.0
SET P0106 P0006
SFTON P0106
REFP 3 C00043 BC00043
CALL JOB:SEARCH-R1
SET P0106 P0006
SFTON P0106
SFTOF
MOVL C00044 BC00044 V=166.7 PL=0
MOVJ C00045 BC00045 VJ=25.00
MOVJ C00046 BC00046 VJ=25.00
MOVJ C00047 BC00047 VJ=25.00
MOVJ C00048 BC00048 VJ=25.00
'TEST
MOVJ C00049 BC00049 VJ=20.00
SFTOF
'------------------------
'W44 P
'------------------------
'TEST
MOVL C00050 BC00050 V=133.3 PL=0
REFP 3 C00051 BC00051
CALL JOB:SEARCH-R1
IMOV P0057 V=23.0
SET P0107 P0006
SFTON P0107
REFP 3 C00052 BC00052
CALL JOB:SEARCH-R1
SET P0107 P0006
SFTON P0107
SFTOF
MOVL C00053 BC00053 V=250.0 PL=0
'TEST
MOVL C00054 BC00054 V=416.7
MOVL C00055 BC00055 V=166.7 PL=0
REFP 3 C00056 BC00056
CALL JOB:SEARCH-R1
IMOV P0057 V=23.0
SET P0108 P0006
SFTON P0108
REFP 3 C00057 BC00057
CALL JOB:SEARCH-R1
SET P0108 P0006
SFTON P0108
SFTOF
MOVL C00058 BC00058 V=250.0 PL=0
'TEST
SFTOF
MOVL C00059 BC00059 V=250.0
MOVJ C00060 BC00060 VJ=25.00
CALL JOB:FRONT_SEARCH_0ST-2_4040_V2
MOVJ C00061 BC00061 VJ=40.00
MOVJ C00062 BC00062 VJ=40.00
MOVJ C00063 BC00063 VJ=40.00
'WELD
'WELD
MOVJ C00064 BC00064 VJ=20.00
'**********************
'W36
'**********************
MOVL C00065 BC00065 V=500.0
SFTON P0105
MOVL C00066 BC00066 V=166.7 PL=0
SFTOF
MACRO1 MJ#(0) ARGF24
ARCON
SFTON P0106
MOVL C00067 BC00067 V=11.0
ARCOF
SFTOF
MOVJ C00068 BC00068 VJ=15.00
MOVJ C00069 BC00069 VJ=30.00
MOVJ C00070 BC00070 VJ=10.00
MOVJ C00071 BC00071 VJ=10.00
MOVJ C00072 BC00072 VJ=30.00
MOVJ C00073 BC00073 VJ=20.00
MOVJ C00074 BC00074 VJ=10.00
MOVJ C00075 BC00075 VJ=15.00
'**********************
'W38
'**********************
MOVL C00076 BC00076 V=500.0
SFTON P0100
MOVL C00077 BC00077 V=166.7 PL=0
SFTOF
ARCON
SFTON P0099
MOVL C00078 BC00078 V=11.0
ARCOF
SFTOF
'DODANE
MOVL C00079 BC00079 V=500.0
MOVL C00080 BC00080 V=666.7
MOVJ C00081 BC00081 VJ=10.00
MOVJ C00082 BC00082 VJ=10.00
MOVJ C00083 BC00083 VJ=10.00
MOVJ C00084 BC00084 VJ=10.00
MOVJ C00085 BC00085 VJ=25.00
MOVJ C00086 BC00086 VJ=30.00
MOVJ C00087 BC00087 VJ=25.00
MOVJ C00088 BC00088 VJ=30.00
MOVJ C00089 BC00089 VJ=30.00
MOVL C00090 BC00090 V=500.0
SFTON P0108
MOVL C00091 BC00091 V=166.7 PL=0
MACRO1 MJ#(0) ARGF24
ARCON
MOVL C00092 BC00092 V=10.8
SFTON P0107
MOVL C00093 BC00093 V=10.8
MOVL C00094 BC00094 V=10.8
ARCOF
SFTOF
MOVL C00095 BC00095 V=500.0
MOVL C00096 BC00096 V=500.0
MOVJ C00097 BC00097 VJ=30.00
'**********************
'W45
'**********************
MOVJ C00098 BC00098 VJ=30.00
MOVJ C00099 BC00099 VJ=20.00
MOVJ C00100 BC00100 VJ=10.00
MACRO1 MJ#(0) ARGF24
MOVL C00101 BC00101 V=500.0
SFTON P0102
MOVL C00102 BC00102 V=166.7 PL=0
ARCON
SFTON P0101
MOVL C00103 BC00103 V=12.5
ARCOF
SFTOF
MOVL C00104 BC00104 V=500.0
'DODANE
MOVJ C00105 BC00105 VJ=10.00
'**********************
'W48
'**********************
MOVJ C00106 BC00106 VJ=15.00
MOVJ C00107 BC00107 VJ=25.00
MOVJ C00108 BC00108 VJ=15.00
SFTON P0104
MOVL C00109 BC00109 V=166.7 PL=0
ARCON
SFTON P0103
MOVL C00110 BC00110 V=10.5
ARCOF
SFTOF
MOVL C00111 BC00111 V=500.0
MOVJ C00112 BC00112 VJ=40.00
CALL JOB:FRONT_WELD_0ST-2_4040_V2
CALL JOB:MOVE_OUT_OF_TUNNEL
CALL JOB:CLEAN-R1
CALL JOB:MOVE_INTO_TUNNEL
MOVJ C00113 BC00113 VJ=30.00 PL=0
'------------------------
'------------------------
'PRAWA STRONA PROFIL GORA
'------------------------
'------------------------
MOVJ C00114 BC00114 VJ=20.00
'------------------------
'W51A L
'------------------------
SFTOF
MOVJ C00115 BC00115 VJ=10.00
MOVL C00116 BC00116 V=66.7 PL=0
REFP 3 C00117 BC00117
CALL JOB:SEARCH-R1
SET P0299 P0006
SFTON P0299
MOVL C00118 BC00118 V=66.7 PL=0
REFP 3 C00119 BC00119
CALL JOB:SEARCH-R1
SET P0299 P0006
SFTON P0299
MOVL C00120 BC00120 V=83.3
MOVL C00121 BC00121 V=166.7 PL=0
REFP 3 C00122 BC00122
CALL JOB:SEARCH-R1
SET P0299 P0006
SFTON P0299
MOVL C00123 BC00123 V=133.3 PL=0
SFTOF
'------------------------
'W51A P
'------------------------
SFTOF
MOVL C00124 BC00124 V=250.0
'------------------------
'W54A L
'------------------------
SFTOF
MOVJ C00125 BC00125 VJ=30.00
MOVL C00126 BC00126 V=133.3 PL=0
REFP 3 C00127 BC00127
CALL JOB:SEARCH-R1
SET P0301 P0006
SFTON P0301
MOVL C00128 BC00128 V=66.7 PL=0
REFP 3 C00129 BC00129
CALL JOB:SEARCH-R1
SET P0301 P0006
SFTON P0301
MOVL C00130 BC00130 V=66.7 PL=0
SFTOF
'------------------------
'W54A P
'------------------------
SFTOF
MOVJ C00131 BC00131 VJ=30.00
MOVL C00132 BC00132 V=133.3 PL=0
REFP 3 C00133 BC00133
CALL JOB:SEARCH-R1
SET P0302 P0006
SFTON P0302
MOVL C00134 BC00134 V=66.7 PL=0
REFP 3 C00135 BC00135
CALL JOB:SEARCH-R1
SET P0302 P0006
SFTON P0302
MOVL C00136 BC00136 V=66.7 PL=0
SFTOF
'------------------------
'W50A L
'------------------------
SFTOF
MOVJ C00137 BC00137 VJ=30.00
MOVL C00138 BC00138 V=133.3 PL=0
REFP 3 C00139 BC00139
CALL JOB:SEARCH-R1
SET P0303 P0006
SFTON P0303
MOVL C00140 BC00140 V=66.7 PL=0
REFP 3 C00141 BC00141
CALL JOB:SEARCH-R1
SET P0303 P0006
SFTON P0303
MOVL C00142 BC00142 V=66.7 PL=0
SFTOF
'------------------------
'W50A P
'------------------------
SFTOF
MOVJ C00143 BC00143 VJ=30.00
MOVL C00144 BC00144 V=133.3 PL=0
REFP 3 C00145 BC00145
CALL JOB:SEARCH-R1
SET P0304 P0006
SFTON P0304
MOVL C00146 BC00146 V=66.7 PL=0
REFP 3 C00147 BC00147
CALL JOB:SEARCH-R1
SET P0304 P0006
SFTON P0304
MOVL C00148 BC00148 V=66.7 PL=0
SFTOF
'------------------------
'W53A L
'------------------------
SFTOF
MOVJ C00149 BC00149 VJ=30.00
MOVL C00150 BC00150 V=133.3 PL=0
REFP 3 C00151 BC00151
CALL JOB:SEARCH-R1
SET P0305 P0006
SFTON P0305
MOVL C00152 BC00152 V=66.7 PL=0
REFP 3 C00153 BC00153
CALL JOB:SEARCH-R1
SET P0305 P0006
SFTON P0305
MOVL C00154 BC00154 V=66.7 PL=0
SFTOF
'------------------------
'W53A P
'------------------------
SFTOF
MOVJ C00155 BC00155 VJ=30.00
MOVL C00156 BC00156 V=200.0
MOVL C00157 BC00157 V=66.7 PL=0
REFP 3 C00158 BC00158
CALL JOB:SEARCH-R1
SET P0306 P0006
SFTON P0306
MOVL C00159 BC00159 V=66.7 PL=0
REFP 3 C00160 BC00160
CALL JOB:SEARCH-R1
SET P0306 P0006
SFTON P0306
MOVL C00161 BC00161 V=66.7 PL=0
SFTOF
'------------------------
'W56A L
'------------------------
SFTOF
MOVJ C00162 BC00162 VJ=30.00
MOVL C00163 BC00163 V=133.3 PL=0
REFP 3 C00164 BC00164
CALL JOB:SEARCH-R1
SET P0307 P0006
SFTON P0307
MOVL C00165 BC00165 V=66.7 PL=0
REFP 3 C00166 BC00166
CALL JOB:SEARCH-R1
SET P0307 P0006
SFTON P0307
MOVL C00167 BC00167 V=66.7 PL=0
SFTOF
'------------------------
'W56A P
'------------------------
SFTOF
MOVJ C00168 BC00168 VJ=30.00
MOVL C00169 BC00169 V=133.3 PL=0
REFP 3 C00170 BC00170
CALL JOB:SEARCH-R1
SET P0308 P0006
SFTON P0308
MOVL C00171 BC00171 V=66.7 PL=0
REFP 3 C00172 BC00172
CALL JOB:SEARCH-R1
SET P0308 P0006
SFTON P0308
MOVL C00173 BC00173 V=66.7 PL=0
SFTOF
'------------------------
COMM SFTOF
COMM MOVJ C00174 BC00174 VJ=30.00
COMM MOVL C00175 BC00175 V=250.0
COMM MOVL C00176 BC00176 V=66.7 PL=0
COMM REFP 3 C00177 BC00177
COMM CALL JOB:SEARCH-R1
COMM SET P0309 P0006
COMM SFTON P0309
COMM MOVL C00178 BC00178 V=66.7 PL=0
COMM REFP 3 C00179 BC00179
COMM CALL JOB:SEARCH-R1
COMM SET P0309 P0006
COMM SFTON P0309
COMM MOVL C00180 BC00180 V=66.7 PL=0
COMM SFTOF
COMM '------------------------
COMM SFTOF
COMM MOVJ C00181 BC00181 VJ=5.00
COMM MOVJ C00182 BC00182 VJ=20.00
COMM MOVL C00183 BC00183 V=116.7 PL=0
COMM REFP 3 C00184 BC00184
COMM CALL JOB:SEARCH-R1
COMM SET P0310 P0006
COMM SFTON P0310
COMM MOVL C00185 BC00185 V=66.7 PL=0
COMM REFP 3 C00186 BC00186
COMM CALL JOB:SEARCH-R1
COMM SET P0310 P0006
COMM SFTON P0310
COMM MOVL C00187 BC00187 V=66.7 PL=0
COMM SFTOF
COMM '------------------------
COMM 'W55A L
COMM '------------------------
SFTOF
MOVL C00188 BC00188 V=250.0
MOVJ C00189 BC00189 VJ=10.00
MOVL C00190 BC00190 V=66.7 PL=0
REFP 3 C00191 BC00191
CALL JOB:SEARCH-R1
SET P0309 P0006
SFTON P0309
MOVL C00192 BC00192 V=66.7 PL=0
REFP 3 C00193 BC00193
CALL JOB:SEARCH-R1
SET P0309 P0006
SFTON P0309
MOVL C00194 BC00194 V=66.7 PL=0
SFTOF
'------------------------
'W55A P
'------------------------
SFTOF
MOVL C00195 BC00195 V=250.0
MOVL C00196 BC00196 V=166.7
MOVL C00197 BC00197 V=66.7 PL=0
REFP 3 C00198 BC00198
CALL JOB:SEARCH-R1
SET P0310 P0006
SFTON P0310
MOVL C00199 BC00199 V=66.7 PL=0
REFP 3 C00200 BC00200
CALL JOB:SEARCH-R1
SET P0310 P0006
SFTON P0310
MOVL C00201 BC00201 V=66.7 PL=0
MOVL C00202 BC00202 V=166.7
SFTOF
MOVL C00203 BC00203 V=250.0
MOVJ C00204 BC00204 VJ=20.00
MOVJ C00205 BC00205 VJ=30.00
MOVJ C00206 BC00206 VJ=20.00
MOVJ C00207 BC00207 VJ=20.00
MOVJ C00208 BC00208 VJ=20.00
MOVJ C00209 BC00209 VJ=20.00
MOVJ C00210 BC00210 VJ=20.00
'------------------------
'LEWA STRONA PROFIL GORA
'------------------------
MOVJ C00211 BC00211 VJ=10.00
'------------------------
SFTOF
MOVJ C00212 BC00212 VJ=10.00
MOVL C00213 BC00213 V=66.7 PL=0
REFP 3 C00214 BC00214
CALL JOB:SEARCH-R1
SET P0351 P0006
SFTON P0351
MOVL C00215 BC00215 V=66.7 PL=0
REFP 3 C00216 BC00216
CALL JOB:SEARCH-R1
SET P0351 P0006
SFTON P0351
MOVL C00217 BC00217 V=66.7 PL=0
SFTOF
MOVJ C00218 BC00218 VJ=10.00
MOVJ C00219 BC00219 VJ=10.00
'------------------------
'W55B P
'------------------------
SFTOF
MOVL C00220 BC00220 V=66.7 PL=0
REFP 3 C00221 BC00221
CALL JOB:SEARCH-R1
SET P0352 P0006
SFTON P0352
MOVL C00222 BC00222 V=66.7 PL=0
REFP 3 C00223 BC00223
CALL JOB:SEARCH-R1
SET P0352 P0006
SFTON P0352
MOVL C00224 BC00224 V=66.7 PL=0
SFTOF
'------------------------
'W52B L
'------------------------
SFTOF
MOVJ C00225 BC00225 VJ=20.00
COMM MOVJ C00226 BC00226 VJ=20.00
COMM MOVL C00227 BC00227 V=150.0
COMM MOVL C00228 BC00228 V=66.7 PL=0
COMM REFP 3 C00229 BC00229
COMM CALL JOB:SEARCH-R1
COMM SET P0351 P0006
COMM SFTON P0351
COMM MOVL C00230 BC00230 V=66.7 PL=0
COMM REFP 3 C00231 BC00231
COMM CALL JOB:SEARCH-R1
COMM SET P0351 P0006
COMM SFTON P0351
COMM MOVL C00232 BC00232 V=66.7 PL=0
COMM SFTOF
COMM '------------------------
COMM 'W52B P
COMM '------------------------
COMM SFTOF
COMM MOVJ C00233 BC00233 VJ=30.00
COMM MOVL C00234 BC00234 V=116.7 PL=0
COMM REFP 3 C00235 BC00235
COMM CALL JOB:SEARCH-R1
COMM SET P0352 P0006
COMM SFTON P0352
COMM MOVL C00236 BC00236 V=66.7 PL=0
COMM REFP 3 C00237 BC00237
COMM CALL JOB:SEARCH-R1
COMM SET P0352 P0006
COMM SFTON P0352
COMM MOVL C00238 BC00238 V=66.7 PL=0
COMM SFTOF
COMM '------------------------
COMM 'W56B L
COMM '------------------------
COMM SFTOF
MOVJ C00239 BC00239 VJ=30.00
MOVL C00240 BC00240 V=116.7 PL=0
REFP 3 C00241 BC00241
CALL JOB:SEARCH-R1
SET P0353 P0006
SFTON P0353
MOVL C00242 BC00242 V=66.7 PL=0
REFP 3 C00243 BC00243
CALL JOB:SEARCH-R1
SET P0353 P0006
SFTON P0353
MOVL C00244 BC00244 V=66.7 PL=0
SFTOF
'------------------------
'W56B P
'------------------------
SFTOF
MOVJ C00245 BC00245 VJ=30.00
MOVL C00246 BC00246 V=116.7 PL=0
REFP 3 C00247 BC00247
CALL JOB:SEARCH-R1
SET P0354 P0006
SFTON P0354
MOVL C00248 BC00248 V=66.7 PL=0
REFP 3 C00249 BC00249
CALL JOB:SEARCH-R1
SET P0354 P0006
SFTON P0354
MOVL C00250 BC00250 V=66.7 PL=0
SFTOF
'------------------------
'W53B L
'------------------------
SFTOF
MOVJ C00251 BC00251 VJ=30.00
MOVL C00252 BC00252 V=116.7 PL=0
REFP 3 C00253 BC00253
CALL JOB:SEARCH-R1
SET P0355 P0006
SFTON P0355
MOVL C00254 BC00254 V=66.7 PL=0
REFP 3 C00255 BC00255
CALL JOB:SEARCH-R1
SET P0355 P0006
SFTON P0355
MOVL C00256 BC00256 V=66.7 PL=0
SFTOF
'------------------------
'W53B P
'------------------------
SFTOF
MOVJ C00257 BC00257 VJ=30.00
MOVL C00258 BC00258 V=116.7 PL=0
REFP 3 C00259 BC00259
CALL JOB:SEARCH-R1
SET P0356 P0006
SFTON P0356
MOVL C00260 BC00260 V=66.7 PL=0
REFP 3 C00261 BC00261
CALL JOB:SEARCH-R1
SET P0356 P0006
SFTON P0356
MOVL C00262 BC00262 V=66.7 PL=0
SFTOF
'------------------------
'W50B L
'------------------------
SFTOF
MOVJ C00263 BC00263 VJ=30.00
MOVL C00264 BC00264 V=116.7 PL=0
REFP 3 C00265 BC00265
CALL JOB:SEARCH-R1
SET P0357 P0006
SFTON P0357
MOVL C00266 BC00266 V=66.7 PL=0
REFP 3 C00267 BC00267
CALL JOB:SEARCH-R1
SET P0357 P0006
SFTON P0357
MOVL C00268 BC00268 V=66.7 PL=0
SFTOF
'------------------------
'W50B P
'------------------------
SFTOF
MOVJ C00269 BC00269 VJ=30.00
MOVL C00270 BC00270 V=116.7 PL=0
REFP 3 C00271 BC00271
CALL JOB:SEARCH-R1
SET P0358 P0006
SFTON P0358
MOVL C00272 BC00272 V=66.7 PL=0
REFP 3 C00273 BC00273
CALL JOB:SEARCH-R1
SET P0358 P0006
SFTON P0358
MOVL C00274 BC00274 V=66.7 PL=0
SFTOF
'------------------------
'W54B L
'------------------------
SFTOF
MOVJ C00275 BC00275 VJ=30.00
MOVL C00276 BC00276 V=116.7 PL=0
REFP 3 C00277 BC00277
CALL JOB:SEARCH-R1
SET P0359 P0006
SFTON P0359
MOVL C00278 BC00278 V=66.7 PL=0
REFP 3 C00279 BC00279
CALL JOB:SEARCH-R1
SET P0359 P0006
SFTON P0359
MOVL C00280 BC00280 V=66.7 PL=0
SFTOF
'------------------------
'W54B P
'------------------------
SFTOF
MOVJ C00281 BC00281 VJ=30.00
MOVL C00282 BC00282 V=116.7 PL=0
REFP 3 C00283 BC00283
CALL JOB:SEARCH-R1
SET P0360 P0006
SFTON P0360
MOVL C00284 BC00284 V=66.7 PL=0
REFP 3 C00285 BC00285
CALL JOB:SEARCH-R1
SET P0360 P0006
SFTON P0360
MOVL C00286 BC00286 V=166.7 PL=0
SFTOF
'------------------------
'W51B L
'------------------------
'------------------------
SFTOF
MOVL C00287 BC00287 V=150.0
MOVL C00288 BC00288 V=66.7 PL=0
REFP 3 C00289 BC00289
CALL JOB:SEARCH-R1
SET P0361 P0006
SFTON P0361
MOVL C00290 BC00290 V=66.7 PL=0
REFP 3 C00291 BC00291
CALL JOB:SEARCH-R1
SET P0361 P0006
SFTON P0361
MOVL C00292 BC00292 V=83.3
MOVL C00293 BC00293 V=133.3 PL=0
REFP 3 C00294 BC00294
CALL JOB:SEARCH-R1
SET P0361 P0006
SFTON P0361
SFTOF
MOVL C00295 BC00295 V=83.3
MOVJ C00296 BC00296 VJ=20.00
MOVJ C00297 BC00297 VJ=30.00
MOVJ C00298 BC00298 VJ=10.00
MOVJ C00299 BC00299 VJ=40.00
'**********************
'**********************
'POCZATEK SPAWANIA BOKI
'**********************
'**********************
MOVJ C00300 BC00300 VJ=30.00
MOVJ C00301 BC00301 VJ=20.00
'**********************
'W50A
'**********************
MOVL C00302 BC00302 V=250.0
SFTON P0304
MOVL C00303 BC00303 V=83.3 PL=0
SFTOF
MACRO1 MJ#(0) ARGF10
ARCON
SFTON P0303
MOVL C00304 BC00304 V=10.8
ARCOF
SFTOF
MOVL C00305 BC00305 V=250.0
'W13B
MOVJ C00306 BC00306 VJ=20.00
MOVJ C00307 BC00307 VJ=40.00
MOVJ C00308 BC00308 VJ=20.00
MOVJ C00309 BC00309 VJ=20.00
MOVJ C00310 BC00310 VJ=20.00
'**********************
'W50B
'**********************
MOVL C00311 BC00311 V=250.0
SFTON P0357
MOVL C00312 BC00312 V=166.7 PL=0
SFTOF
MACRO1 MJ#(0) ARGF10
ARCON
SFTON P0358
MOVL C00313 BC00313 V=10.8
ARCOF
SFTOF
MOVL C00314 BC00314 V=250.0
MOVJ C00315 BC00315 VJ=20.00
MOVJ C00316 BC00316 VJ=20.00
MOVJ C00317 BC00317 VJ=20.00
MOVJ C00318 BC00318 VJ=20.00
'**********************
'W51A
'**********************
MOVL C00319 BC00319 V=416.7
SFTON P0299
MOVL C00320 BC00320 V=166.7 PL=0
SFTOF
MACRO1 MJ#(0) ARGF10
ARCON
SFTON P0299
MOVL C00321 BC00321 V=10.8
MOVL C00322 BC00322 V=10.8
ARCOF
MOVL C00323 BC00323 V=166.7
MOVL C00324 BC00324 V=133.3 PL=0
ARCON
MOVL C00325 BC00325 V=8.3
ARCOF
SFTOF
MOVL C00326 BC00326 V=200.0
MOVJ C00327 BC00327 VJ=30.00
MOVJ C00328 BC00328 VJ=30.00
MOVJ C00329 BC00329 VJ=30.00
MOVJ C00330 BC00330 VJ=30.00
MOVJ C00331 BC00331 VJ=30.00
'**********************
'W51B
'**********************
MOVL C00332 BC00332 V=416.7
MOVL C00333 BC00333 V=416.7
SFTON P0361
MOVL C00334 BC00334 V=166.7 PL=0
SFTOF
MACRO1 MJ#(0) ARGF10
ARCON
SFTON P0361
MOVL C00335 BC00335 V=10.8
MOVL C00336 BC00336 V=10.8
ARCOF
MOVL C00337 BC00337 V=166.7
MACRO1 MJ#(0) ARGF9
MOVL C00338 BC00338 V=166.7 PL=0
ARCON
MOVL C00339 BC00339 V=8.3
ARCOF
SFTOF
MOVL C00340 BC00340 V=166.7
MOVL C00341 BC00341 V=250.0
MOVJ C00342 BC00342 VJ=30.00
MOVJ C00343 BC00343 VJ=30.00
MOVJ C00344 BC00344 VJ=30.00
MOVJ C00345 BC00345 VJ=40.00
MOVJ C00346 BC00346 VJ=40.00
MOVJ C00347 BC00347 VJ=20.00
MOVJ C00348 BC00348 VJ=20.00
MOVJ C00349 BC00349 VJ=20.00
MOVJ C00350 BC00350 VJ=20.00
MOVJ C00351 BC00351 VJ=20.00
'**********************
'W52A
'**********************
SFTON P0310
MOVL C00352 BC00352 V=250.0
MOVL C00353 BC00353 V=83.3 PL=0
SFTOF
MACRO1 MJ#(0) ARGF10
ARCON
SFTON P0309
MOVL C00354 BC00354 V=10.8
ARCOF
SFTOF
MOVL C00355 BC00355 V=333.3
MOVJ C00356 BC00356 VJ=30.00
MOVJ C00357 BC00357 VJ=30.00
MOVJ C00358 BC00358 VJ=30.00
MOVJ C00359 BC00359 VJ=30.00
MOVJ C00360 BC00360 VJ=30.00
MOVJ C00361 BC00361 VJ=20.00
MOVJ C00362 BC00362 VJ=20.00
MOVJ C00363 BC00363 VJ=20.00
'**********************
'52B
'**********************
MOVL C00364 BC00364 V=250.0
SFTON P0351
MOVL C00365 BC00365 V=83.3 PL=0
MACRO1 MJ#(0) ARGF10
ARCON
SFTON P0352
MOVL C00366 BC00366 V=10.8
ARCOF
MOVL C00367 BC00367 V=333.3
SFTOF
MOVJ C00368 BC00368 VJ=20.00
MOVJ C00369 BC00369 VJ=30.00
MOVJ C00370 BC00370 VJ=30.00
'**********************
'W53A
'**********************
MOVJ C00371 BC00371 VJ=30.00
MOVJ C00372 BC00372 VJ=30.00
MOVJ C00373 BC00373 VJ=10.00
'**********************
'W53A
'**********************
SFTON P0306
MOVL C00374 BC00374 V=250.0
MOVL C00375 BC00375 V=83.3 PL=0
SFTOF
MACRO1 MJ#(0) ARGF10
ARCON
SFTON P0305
MOVL C00376 BC00376 V=10.8
ARCOF
SFTOF
MOVL C00377 BC00377 V=250.0
MOVJ C00378 BC00378 VJ=30.00
MOVJ C00379 BC00379 VJ=30.00
MOVJ C00380 BC00380 VJ=30.00
MOVJ C00381 BC00381 VJ=30.00
MOVJ C00382 BC00382 VJ=30.00
MOVJ C00383 BC00383 VJ=30.00
MOVL C00384 BC00384 V=250.0
'**********************
'W53B
'**********************
SFTON P0355
MOVL C00385 BC00385 V=250.0
MOVL C00386 BC00386 V=83.3 PL=0
SFTOF
MACRO1 MJ#(0) ARGF10
ARCON
SFTON P0356
MOVL C00387 BC00387 V=10.8
ARCOF
SFTOF
MOVL C00388 BC00388 V=333.3
MOVJ C00389 BC00389 VJ=30.00
MOVJ C00390 BC00390 VJ=30.00
MOVJ C00391 BC00391 VJ=30.00
MOVJ C00392 BC00392 VJ=30.00
'**********************
'W54A
'**********************
SFTON P0302
MOVL C00393 BC00393 V=250.0
MOVL C00394 BC00394 V=83.3 PL=0
SFTOF
MACRO1 MJ#(0) ARGF10
ARCON
SFTON P0301
MOVL C00395 BC00395 V=10.8
ARCOF
SFTOF
MOVL C00396 BC00396 V=333.3
MOVJ C00397 BC00397 VJ=20.00
MOVJ C00398 BC00398 VJ=30.00
MOVJ C00399 BC00399 VJ=30.00
MOVJ C00400 BC00400 VJ=30.00
MOVJ C00401 BC00401 VJ=30.00
'**********************
'W54B
'**********************
SFTON P0359
MOVL C00402 BC00402 V=250.0
MOVL C00403 BC00403 V=83.3 PL=0
SFTOF
MACRO1 MJ#(0) ARGF10
ARCON
SFTON P0360
MOVL C00404 BC00404 V=10.8
ARCOF
MOVL C00405 BC00405 V=333.3
SFTOF
MOVJ C00406 BC00406 VJ=30.00
MOVJ C00407 BC00407 VJ=30.00
MOVJ C00408 BC00408 VJ=30.00
MOVJ C00409 BC00409 VJ=40.00
MOVJ C00410 BC00410 VJ=40.00
COMM MOVJ C00411 BC00411 VJ=10.00
COMM MOVJ C00412 BC00412 VJ=10.00
COMM MOVJ C00413 BC00413 VJ=10.00
COMM MOVJ C00414 BC00414 VJ=15.00
COMM MOVJ C00415 BC00415 VJ=15.00
COMM MOVJ C00416 BC00416 VJ=15.00
COMM MOVJ C00417 BC00417 VJ=15.00
COMM '**********************
COMM 'W55A
COMM '**********************
COMM SFTON P0311
COMM MOVL C00418 BC00418 V=166.7 PL=0
COMM SFTOF
COMM MACRO1 MJ#(0) ARGF10
COMM ARCON
COMM SFTON P0312
COMM MOVL C00419 BC00419 V=10.8
COMM MOVL C00420 BC00420 V=10.8
COMM ARCOF
COMM SFTOF
COMM MOVL C00421 BC00421 V=150.0
COMM MOVJ C00422 BC00422 VJ=10.00
COMM MOVJ C00423 BC00423 VJ=10.00
COMM MOVJ C00424 BC00424 VJ=10.00
COMM MOVJ C00425 BC00425 VJ=10.00
COMM MOVJ C00426 BC00426 VJ=10.00
COMM MOVJ C00427 BC00427 VJ=10.00
COMM MOVJ C00428 BC00428 VJ=30.00
COMM MOVJ C00429 BC00429 VJ=30.00
COMM MOVJ C00430 BC00430 VJ=20.00
COMM MOVJ C00431 BC00431 VJ=30.00
COMM MOVJ C00432 BC00432 VJ=20.00
COMM MOVJ C00433 BC00433 VJ=20.00
COMM MOVJ C00434 BC00434 VJ=30.00
COMM MOVJ C00435 BC00435 VJ=20.00
COMM MOVJ C00436 BC00436 VJ=20.00
COMM '**********************
COMM 'W55B
COMM '**********************
COMM SFTON P0350
COMM MOVL C00437 BC00437 V=333.3
COMM MOVL C00438 BC00438 V=166.7 PL=0
COMM SFTOF
COMM MACRO1 MJ#(0) ARGF10
COMM ARCON
COMM SFTON P0349
COMM MOVL C00439 BC00439 V=10.8
COMM MOVL C00440 BC00440 V=10.8
COMM ARCOF
COMM SFTOF
COMM MOVL C00441 BC00441 V=66.7
COMM MOVJ C00442 BC00442 VJ=10.00
COMM MOVJ C00443 BC00443 VJ=20.00
COMM MOVJ C00444 BC00444 VJ=20.00
COMM MOVJ C00445 BC00445 VJ=20.00
MOVJ C00446 BC00446 VJ=30.00
MOVJ C00447 BC00447 VJ=50.00
MOVJ C00448 BC00448 VJ=50.00
MOVJ C00449 BC00449 VJ=40.00
MOVJ C00450 BC00450 VJ=20.00
'**********************
'W56A
'**********************
SFTON P0308
MOVL C00451 BC00451 V=333.3
MOVL C00452 BC00452 V=166.7 PL=0
SFTOF
MACRO1 MJ#(0) ARGF10
ARCON
SFTON P0307
MOVL C00453 BC00453 V=10.8
ARCOF
SFTOF
MOVL C00454 BC00454 V=333.3
MOVJ C00455 BC00455 VJ=20.00
MOVJ C00456 BC00456 VJ=30.00
MOVJ C00457 BC00457 VJ=30.00
MOVJ C00458 BC00458 VJ=30.00
'**********************
'W56B
'**********************
SFTON P0353
MOVL C00459 BC00459 V=250.0
MOVL C00460 BC00460 V=166.7 PL=0
SFTOF
MACRO1 MJ#(0) ARGF10
ARCON
SFTON P0354
MOVL C00461 BC00461 V=10.8
ARCOF
SFTOF
MOVL C00462 BC00462 V=333.3
MOVJ C00463 BC00463 VJ=30.00
MOVJ C00464 BC00464 VJ=30.00
MOVJ C00465 BC00465 VJ=30.00
CALL JOB:MOVE_OUT_OF_TUNNEL
CALL JOB:R1-HOME
END
